(* IEC 61131-3 sources: crb-codesys/retrieval/output/codesys_repo/电子凸轮运动实训/FUN, 4 files *)

(* ---- F_AxisStatusToString.st ---- *)
FUNCTION F_AxisStatusToString : STRING
VAR_INPUT
	fbReadStatus	:	MC_ReadStatus;		//轴状态读取功能块
END_VAR

// 根据轴状态返回对应的字符串描述
// 按优先级顺序检查状态

IF fbReadStatus.Errorstop THEN
	F_AxisStatusToString := 'Errorstop';
	RETURN;
END_IF

IF fbReadStatus.Disabled THEN
	F_AxisStatusToString := 'Disabled';
	RETURN;
END_IF

IF fbReadStatus.Homing THEN
	F_AxisStatusToString := 'Homing';
	RETURN;
END_IF

IF fbReadStatus.Stopping THEN
	F_AxisStatusToString := 'Stopping';
	RETURN;
END_IF

IF fbReadStatus.SynchronizedMotion THEN
	F_AxisStatusToString := 'SynchronizedMotion';
	RETURN;
END_IF

IF fbReadStatus.ContinuousMotion THEN
	F_AxisStatusToString := 'ContinuousMotion';
	RETURN;
END_IF

IF fbReadStatus.DiscreteMotion THEN
	F_AxisStatusToString := 'DiscreteMotion';
	RETURN;
END_IF

IF fbReadStatus.StandStill THEN
	F_AxisStatusToString := 'StandStill';
	RETURN;
END_IF

// 默认状态
F_AxisStatusToString := 'Unknown';

(* ---- FB_DualAxisPower.st ---- *)
FUNCTION_BLOCK FB_DualAxisPower
VAR_INPUT
	Axis1			:	AXIS_REF;			//轴1引用
	Axis2			:	AXIS_REF;			//轴2引用
	bPowerOn		:	BOOL;				//电源使能信号
END_VAR
VAR_OUTPUT
	bPowerDone		:	BOOL;				//两轴都准备就绪
	bAxis1Ready		:	BOOL;				//轴1准备就绪
	bAxis2Ready		:	BOOL;				//轴2准备就绪
	bError			:	BOOL;				//错误标志
END_VAR
VAR
	fbPower1		:	MC_Power;			//轴1电源控制
	fbPower2		:	MC_Power;			//轴2电源控制
END_VAR

// 执行轴1电源控制
fbPower1(
	Axis := Axis1,
	Enable := TRUE,
	bDriveStart := bPowerOn,
	bRegulatorOn := bPowerOn
);

// 执行轴2电源控制
fbPower2(
	Axis := Axis2,
	Enable := TRUE,
	bDriveStart := bPowerOn,
	bRegulatorOn := bPowerOn
);

// 更新输出状态
bAxis1Ready := fbPower1.Status;
bAxis2Ready := fbPower2.Status;
bPowerDone := fbPower1.Status AND fbPower2.Status;
bError := fbPower1.Error OR fbPower2.Error;

(* ---- FB_DualAxisReset.st ---- *)
FUNCTION_BLOCK FB_DualAxisReset
VAR_INPUT
	Axis1			:	AXIS_REF;			//轴1引用
	Axis2			:	AXIS_REF;			//轴2引用
	bExecute		:	BOOL;				//执行复位信号
END_VAR
VAR_OUTPUT
	bDone			:	BOOL;				//复位完成
	bBusy			:	BOOL;				//复位进行中
	bError			:	BOOL;				//错误标志
END_VAR
VAR
	fbReset1		:	MC_Reset;			//轴1复位
	fbReset2		:	MC_Reset;			//轴2复位
	fbReadStatus1	:	MC_ReadStatus;		//轴1状态读取
	fbReadStatus2	:	MC_ReadStatus;		//轴2状态读取
	bError1			:	BOOL;				//轴1错误标志
	bError2			:	BOOL;				//轴2错误标志
	nState			:	UDINT;				//状态机
END_VAR

CASE nState OF
	0: (* 空闲状态 *)
		bDone := FALSE;
		bBusy := FALSE;

		IF bExecute THEN
			// 初始化
			fbReset1(Axis := Axis1, Execute := FALSE);
			fbReset2(Axis := Axis2, Execute := FALSE);
			fbReadStatus1(Axis := Axis1, Enable := FALSE);
			fbReadStatus2(Axis := Axis2, Enable := FALSE);
			nState := 1;
		END_IF

	1: (* 读取轴状态 *)
		bBusy := TRUE;

		fbReadStatus1(Axis := Axis1, Enable := TRUE);
		fbReadStatus2(Axis := Axis2, Enable := TRUE);

		IF fbReadStatus1.Valid AND fbReadStatus2.Valid THEN
			bError1 := fbReadStatus1.Errorstop;
			bError2 := fbReadStatus2.Errorstop;
			fbReadStatus1(Axis := Axis1, Enable := FALSE);
			fbReadStatus2(Axis := Axis2, Enable := FALSE);
			nState := 2;
		END_IF

	2: (* 执行复位 *)
		fbReset1(Axis := Axis1, Execute := TRUE);
		fbReset2(Axis := Axis2, Execute := TRUE);
		fbReadStatus1(Axis := Axis1, Enable := TRUE);
		fbReadStatus2(Axis := Axis2, Enable := TRUE);

		IF fbReadStatus1.Valid AND fbReadStatus2.Valid THEN
			bError1 := fbReadStatus1.Errorstop;
			bError2 := fbReadStatus2.Errorstop;
			fbReadStatus1(Axis := Axis1, Enable := FALSE);
			fbReadStatus2(Axis := Axis2, Enable := FALSE);

			// 检查是否还有错误
			IF NOT bError1 AND NOT bError2 THEN
				bDone := TRUE;
				bBusy := FALSE;
				nState := 3;
			ELSE
				bError := TRUE;
				bBusy := FALSE;
				nState := 3;
			END_IF
		END_IF

	3: (* 完成状态 *)
		IF NOT bExecute THEN
			bDone := FALSE;
			bError := FALSE;
			nState := 0;
		END_IF
END_CASE

(* ---- ResetAxis.st ---- *)
FUNCTION_BLOCK ResetAxis
VAR_INPUT
	bExec	:	BOOL;
END_VAR
VAR
	fbReset1	:	MC_Reset;
	fbReset2	:	MC_Reset;

	fbReadAxisError1	:	MC_ReadAxisError;
	fbReadAxisError2	:	MC_ReadAxisError;

	fbReadStatus1	:	MC_ReadStatus;
	fbReadStatus2	:	MC_ReadStatus;

	fbExecTrig	:	R_TRIG;
	nState 	:	BYTE;

	bErrorX	:	BOOL;
	bErrorY	:	BOOL;

END_VAR

VAR_OUTPUT
	Done	:	BOOL;
END_VAR

fbExecTrig(CLK := bExec);

CASE nState OF
	0:
		IF fbExecTrig.Q THEN
			nState := 1;
			Done := FALSE;
		END_IF
	1:
		fbReadAxisError1(Axis := AxisX ,Enable := TRUE);
		fbReadAxisError2(Axis := AxisY ,Enable := TRUE);

		fbReadStatus1(Axis := AxisX ,Enable := TRUE);
		fbReadStatus2(Axis := AxisY ,Enable := TRUE);

		IF fbReadAxisError1.Valid AND fbReadAxisError2.Valid AND fbReadStatus1.Valid AND fbReadStatus2.Valid THEN
			IF fbReadAxisError1.AxisError OR fbReadStatus1.FBErrorOccured THEN
				bErrorX := TRUE;
			ELSE
				bErrorX := FALSE;
			END_IF
			IF fbReadAxisError2.AxisError OR fbReadStatus2.FBErrorOccured THEN
				bErrorY := TRUE;
			ELSE
				bErrorY := FALSE;
			END_IF
			fbReadAxisError1(Axis := AxisX ,Enable := FALSE);
			fbReadAxisError2(Axis := AxisY ,Enable := FALSE);

			fbReadStatus1(Axis := AxisX ,Enable := FALSE);
			fbReadStatus2(Axis := AxisY ,Enable := FALSE);

			fbReset1(Axis := AxisX,Execute := FALSE);
			fbReset2(Axis := AxisY,Execute := FALSE);
			nState := 2;
		END_IF
	2:
		fbReset1(Axis := AxisX,Execute := bErrorX);
		fbReset2(Axis := AxisY,Execute := bErrorY);

		fbReadAxisError1(Axis := AxisX ,Enable := TRUE);
		fbReadAxisError2(Axis := AxisY ,Enable := TRUE);

		fbReadStatus1(Axis := AxisX ,Enable := TRUE);
		fbReadStatus2(Axis := AxisY ,Enable := TRUE);

		IF fbReadAxisError1.Valid AND fbReadAxisError2.Valid AND fbReadStatus1.Valid AND fbReadStatus2.Valid THEN
			IF NOT fbReadAxisError1.AxisError AND NOT fbReadAxisError2.AxisError (* AND NOT fbReadStatus1.FBErrorOccured AND NOT fbReadStatus2.FBErrorOccured AND NOT fbReadStatus3.FBErrorOccured *)THEN
				nState := 0;
				Done := TRUE;

				fbReadAxisError1(Axis := AxisX ,Enable := FALSE);
				fbReadAxisError2(Axis := AxisY ,Enable := FALSE);

				fbReset1(Axis := AxisX,Execute := FALSE);
				fbReset2(Axis := AxisY,Execute := FALSE);

				fbReadStatus1(Axis := AxisX ,Enable := FALSE);
				fbReadStatus2(Axis := AxisY ,Enable := FALSE);
			END_IF
		END_IF
END_CASE
